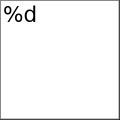
VISUALIZATION VisuStation  // 120x120
VAR_INPUT
	j : INT;
	
END_VAR
    Rectangle (0,0 120x120), "%d", text variable: j
        p3560616238: GVL.StationProcessData[j].VisuPosX
        p2738717112: GVL.iVisuYoffset-GVL.StationProcessData[j].VisuPosY
END_VISUALIZATION

(* stored: Version 1.1.0.1, ProductVersion 3.1.4024.12
   Visu VisuStation: Id {c4fc15e1-0ba4-407f-b7be-e18e9c406fc2} *)
